// TIA Portal V17 export
// export: Created 2025-03-10T13:11:19.9734411Z, ExportSetting WithDefaults, DisplayName Totally Integrated Automation Portal, DisplayVersion V17 Update 8, DisplayName TIA Portal Openness, DisplayVersion V17 Update 8, DisplayName TIA Portal Version Control Interface, DisplayVersion V17, DisplayName SINAMICS Startdrive Advanced, DisplayVersion V17 SP2, DisplayName SINAMICS Startdrive G110M, G120, G120C, G120D, G120P, G115D, DisplayVersion V17 SP2, DisplayName SINAMICS Startdrive G130, G150, S120, S150, SINAMICS MV, S210, DisplayVersion V17 SP2, DisplayName STEP 7 Professional, DisplayVersion V17 Update 8, DisplayName SINUMERIK ONE STEP 7 Toolbox, DisplayVersion V17 Update 12, DisplayName SINUMERIK 840D sl STEP 7 Toolbox, DisplayVersion V17 Update 12, DisplayName STEP 7 Safety, DisplayVersion V17 Update 6, DisplayName WinCC Advanced, DisplayVersion V17 Update 8
DATA_BLOCK "DB2202_DEVSTATE_PROFINET"   // DB2202
{ DB_Accessible_From_OPC_UA := 'FALSE' }
// stored: AutoNumber false, DBAccessibleFromOPCUA false, DBAccessibleFromWebserver true, InstanceOfName LTLP_SLDeviceDiagnostic, InstanceOfType FB
"LTLP_SLDeviceDiagnostic"
   // VAR_INPUT
   //    ID_NETSYSTEM : HW_IOSYSTEM;
   // END_VAR
   // VAR_OUTPUT
   //    RET_VALUE : Word;
   // END_VAR
   // VAR
   //    stDiagnosticData { ExternalAccessible := 'False'; ExternalVisible := 'False'; ExternalWritable := 'False'; S7_SetPoint := 'True'} : "LTLP_typeNetworkDiagnosticState";
   //    stInstGetNameOfDevice { S7_SetPoint := 'True'} : Get_Name;
   //    stInstGeoAddressIOSystem { S7_SetPoint := 'True'} : GEOADDR;
   //    stActualReadCommand : Int;
   //    stActualReadModeDevice : UInt;
   //    stActualReadModeModule : UInt;
   //    stReadDataChanged { ExternalAccessible := 'False'; ExternalVisible := 'False'; ExternalWritable := 'False'} : UInt;
   //    retValueReadConfigured : Int;
   //    retValueReadFailed : Int;
   //    retValueReadDisabled : Int;
   //    retValueReadExists : Int;
   //    retValueReadProblems : Int;
   //    retValueGeo2Log : Int;
   //    allConfiguredDevicesAreRead : Bool;
   //    allExistingDevicesAreRead : Bool;
   //    configuredDevice : Array[0..1023] of Bool;
   //    failedDevice : Array[0..1023] of Bool;
   //    disabledDevice : Array[0..1023] of Bool;
   //    existsDevice : Array[0..1023] of Bool;
   //    hasProblemsDevice : Array[0..1023] of Bool;
   //    geoAddressDevice { S7_SetPoint := 'True'} : GEOADDR;
   // END_VAR
BEGIN
END_DATA_BLOCK
